{region '#Template'}
	{attribute 'Category' := 'Trade'}
	{attribute 'Version' := '0.0.1.0'}
	{attribute 'Tags' := 'Trade, Plant, AC'}
	{attribute 'Description' := 'Aufruf der Anlagen des Gewerks Klimaanlagen	// Calling the plants of the trade air conditioning'}
{endregion}
FUNCTION_BLOCK FB_BA_AC EXTENDS FB_BA_View
VAR_INPUT CONSTANT
AHU01:FB_BA_AHU_1St_PrHtr_ErcPl_Col;
END_VAR
VAR_INPUT
END_VAR
VAR_OUTPUT
END_VAR
VAR
END_VAR

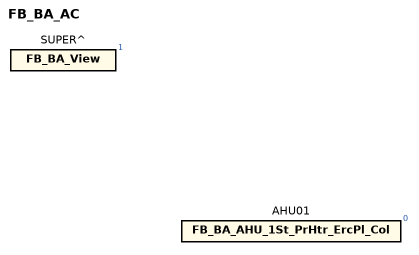
AHU01(); // FB_BA_AHU_1St_PrHtr_ErcPl_Col
SUPER^(); // FB_BA_View

METHOD FB_init : BOOL
VAR_INPUT
	bInitRetains : BOOL; // if TRUE, the retain variables are initialized (warm start / cold start)
	bInCopyCode : BOOL;  // if TRUE, the instance afterwards gets moved into the copy code (online change)
END_VAR
AHU01.iParent 					:= THIS^;	
AHU01.sObjectName				:= CONCAT(TextPlants.Air_handling_unit_sObjectName,'11');											
AHU01.sDescription				:= TextPlants.Air_handling_unit_sDescription;							
AHU01.eDPADMode					:= E_BA_DPADMode.eInclude;

AHU01.GeneralSettings.Subject	:= Site.GeneralSettings_Subject;
AHU01.GeneralSettings.sTarget	:= Site.GeneralSettings_NetId;
END_METHOD

END_FUNCTION_BLOCK

(* stored: Version 1.1.0.1, ProductVersion 3.1.4024.9
   POU FB_BA_AC: Id {f8e80c12-f1b3-4511-8ebc-9fac5dcd318f}, SpecialFunc None
   Method FB_init: Id {c2a7a310-da13-4e69-b20d-dc1ca2ffd44c} *)
